ABB RobotStudio station: Station_[09.05.13]2.rsstn

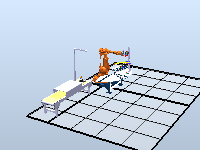
Station Station_[09.05.13] (saved by RobotStudio format 3)
Controller IRB2400_10kg_1.5m_3, task T_ROB1: task frame (RAPID world) sits at (0, 0, 226) mm in the station
Controller IRB2400_10kg_1.5m_3
  mechanical unit ROB_1: IRB2400_10_150__02, 6 joints, base frame (0, 0, -10) mm
Layout (positions relative to the parent item):
  - IRB2400_10_150__02 [mechanism, from Robots\IRB2400_10_150__02.rslib] at (0, 0, 216) mm; joint values [0, 0, 0, 0, 0, 0] (rad or m)
  - Table3_2 [part]
  - SC_RightDispenser [smart component] at (848.89, 660.39, 707) mm, rotated rx 0 ry 0 rz -142.5 deg
      signals: DI diNewPin, DO doPinInPosition2, DO doPinInPosition1
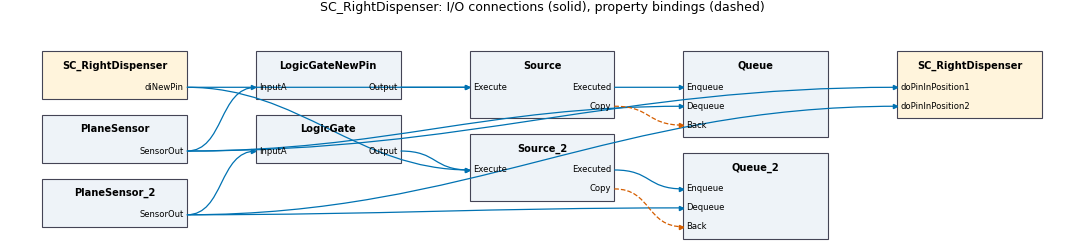
      connections:
        SC_RightDispenser.diNewPin -> Source.Execute
        Source.Executed -> Queue.Enqueue
        PlaneSensor.SensorOut -> Queue.Dequeue
        PlaneSensor.SensorOut -> SC_RightDispenser.doPinInPosition1
        PlaneSensor.SensorOut -> LogicGateNewPin.InputA
        LogicGateNewPin.Output -> Source.Execute
        SC_RightDispenser.diNewPin -> Source_2.Execute
        Source_2.Executed -> Queue_2.Enqueue
        PlaneSensor_2.SensorOut -> Queue_2.Dequeue
        PlaneSensor_2.SensorOut -> SC_RightDispenser.doPinInPosition2
        PlaneSensor_2.SensorOut -> LogicGate.InputA
        LogicGate.Output -> Source_2.Execute
        Source.Copy => Queue.Back
        Source_2.Copy => Queue_2.Back
    - Dispenser [part]
    - Source [smart component]
        properties: Source=Pin; Copy=Pin_291; Parent=(none); Position=[-0.078 0.0985 0.189]; Orientation=[0 0 0]; Transient=false
        signals: DI Execute, DO Executed
    - Queue [smart component]
        properties: Back=Pin_291; Front=(none); Queue={410cd2da-901c-4602-b1b9-b274db1111d8};{51c41708-d6a1-4a4a-81b2-86109b64f340};{5f0a7e8e-897b-4f59-8c9f-8c525d5b29a4};{57ea5d73-423b-4f0f-a570-9931c59fdda0};{5ccf77fa-e120-45a3-9187-0274426f82fc};{74150822-190d-40d8-916f-0fd6875921bc};{baa7ba2a-e563-400f-ae00-338ac9d6b310};{166c1fa7-f084-4893-8c68-a7378bc4935a};{0c8467ce-4cb3-4075-8f36-e6447ecc44ba};{a4931bd6-61c0-4022-957d-34420e4f6ad0};{b2f85a70-4d19-413a-b019-3afa180c1445};{512256d1-278f-462d-98f1-9ffcbd4d9afc};{849db594-4dfe-4c58-a8bd-451d21853566};{c968444c-bd1a-4f2f-bbaa-bfd3e7f50be5};{53c4b951-dfc2-4c08-b51d-efe4876241dc};{64f07cc2-7ba3-4255-a888-147bdde81c96};{5e5e12c0-75f5-4fd7-8049-5710cdd06950};{7bc2919c-0f2a-489c-9e4c-df3bff6561ed};{5aa4b278-0833-4ca9-af8d-253aa8523874};{1baac950-fc54-4ea7-852c-7f888843f6f9};{b4b16473-bd2b-40f5-a110-90fbcba822d9};{d003a69b-5307-4c56-b226-d498155ba824};{d659394f-77c7-41ee-9797-cd61472f6401};{a8294731-aa9f-4324-81a7-55ebbef1ff1c};{1eff712e-2c63-4fa8-99b0-fad1482486d3};{b15f9735-19cd-4f7a-8d4f-e540a16427f5};{02485707-3f80-4cc3-94a6-af0fe382acfb};{ec0e8ce0-b480-4ff5-b740-0a7d244ffb35};{21e78636-7eb3-4061-8dde-926c3e464303};{0772fef3-b80e-464b-9cad-322a585d167a};{d8ed8ead-e522-4938-9c7c-7997e1d5aae1};{4dfefca0-2913-4484-9455-684dfc1cbf5a};{f8c8569f-a97f-4f57-84f0-3da59c0f2755};{9fd95979-e5cf-4fa7-b177-2c560699c82c};{84f56170-3294-4345-a728-b2bfe69be833};{b3710d51-6f0f-48ac-9b0f-811ac7c7d083};{c8300349-23e3-4531-beb4-4210900096fb}; NumberOfObjects=0
        signals: DI Enqueue, DI Dequeue, DI Clear, DI Delete, DI DeleteAll
    - LinearMover [smart component]
        properties: Object=Queue; Direction=[0 0 -0.07]; Speed=0.05; Reference=Global; ReferenceObject=(none)
        signals: DI Execute
    - PlaneSensor [smart component]
        properties: Origin=[-0.0530000000000006 0.1235 0.1195]; Axis1=[-0.03 0 0]; Axis2=[0 -0.04 0]; SensedPart=Pin_291
        signals: DI Active, DO SensorOut
      - _sensorPart_ [part]
    - Pin [part] at (-78, 98.5, 189) mm
    - LogicGateNewPin [smart component]
        properties: Operator=NOT; Delay=0
        signals: DI InputA, DI InputB, DO Output
    - Source_2 [smart component]
        properties: Source=Pin_2; Copy=Pin_2_290; Parent=(none); Position=[-0.078 -0.0985 0.198]; Orientation=[0 0 0]; Transient=false
        signals: DI Execute, DO Executed
    - Queue_2 [smart component]
        properties: Back=Pin_2_290; Front=(none); Queue={9b8a8857-6c8e-4b14-9da2-826ab751c38e};{88bba264-885b-495e-9113-affa9235d31d};{50c1a2e4-cd05-4fea-a5f8-244e054fca82};{1c26a820-5f81-4fc8-b661-270a696b215b};{079caa1e-4b65-4731-ac2d-b38991013e84};{04249497-c8e4-4d2b-8d23-0d0c3b1232f2};{9b46111e-8043-4ec7-820f-f6b1f3216e0a};{190405bf-72c0-4a75-968d-0e05791ba659};{cdaa2867-23d2-4f9c-8306-ddafce1e9ac9};{a0d1b5cc-bcdc-4e7d-b91f-09bc5bc174e5};{802900b3-44c0-4e10-9d61-adfd75a0d86d};{e1828195-6a4a-4e48-b78f-f1287aff9cdc};{27d5d252-1980-452a-aff5-49173c411714};{b44ede4c-8dd3-43ce-8da4-3f1fb091dc7f};{168b000f-829e-439e-a2b5-5bc5735400ce};{aacdfd62-2178-4132-b345-2cd6db76197d};{33bd895a-7dcf-445c-8a77-0a7b01e583dc};{c1a42cbc-38c3-48e5-a615-b149ac9d8780};{fcea76f5-b349-47ef-a520-1d1e9307533b};{d936eec8-07d3-4a18-b33b-be549f4009da};{161ff837-8ce6-447d-8217-59dc5e5add53}; NumberOfObjects=0
        signals: DI Enqueue, DI Dequeue, DI Clear, DI Delete, DI DeleteAll
    - LinearMover_2 [smart component]
        properties: Object=Queue_2; Direction=[0 0 -0.07]; Speed=0.05; Reference=Global; ReferenceObject=(none)
        signals: DI Execute
    - PlaneSensor_2 [smart component]
        properties: Origin=[-0.053 -0.1235 0.1195]; Axis1=[-0.03 0 0]; Axis2=[0 0.04 0]; SensedPart=Pin_2_290
        signals: DI Active, DO SensorOut
      - _sensorPart_ [part]
    - LogicGate [smart component]
        properties: Operator=NOT; Delay=0
        signals: DI InputA, DI InputB, DO Output
    - Pin_2 [part] at (-78, -98.5, 189) mm
    - Pin_2_290 [part] at (-78, -98.5, 118.8) mm
    - Pin_291 [part] at (-78, 98.5, 119.4) mm
  - SC_Conveyor[190413] [smart component] at (45.5, -3634, 0) mm
      signals: DI diPalletOut, DI diPalletIn, DO doPalletAtEnd, DO doPalletAtStart, DO diPalletMovingOut, DO doPalletMovingIn, DI diConDir, DI diConRun
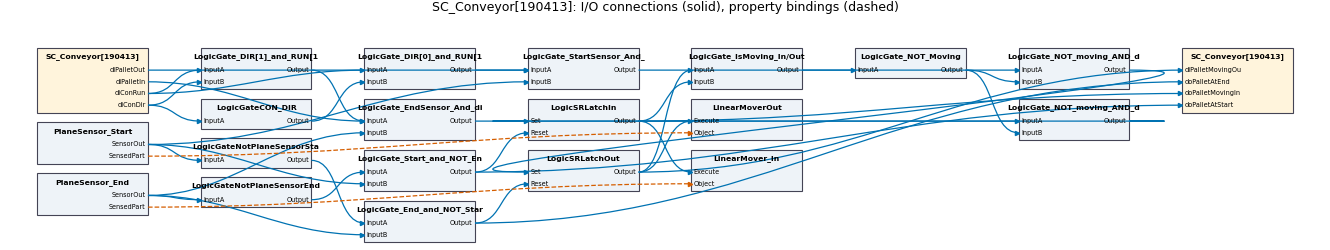
      connections:
        SC_Conveyor[190413].diPalletOut -> LogicGate_StartSensor_And_diOUT.InputA
        PlaneSensor_Start.SensorOut -> LogicGate_StartSensor_And_diOUT.InputB
        PlaneSensor_Start.SensorOut -> LogicGateNotPlaneSensorStart.InputA
        LogicGate_StartSensor_And_diOUT.Output -> LogicGate_NOT_moving_AND_diOUT.InputA
        LogicGate_NOT_Moving.Output -> LogicGate_NOT_moving_AND_diOUT.InputB
        LogicGate_NOT_moving_AND_diOUT.Output -> LogicSRLatchOut.Set
        LogicSRLatchOut.Output -> LinearMoverOut.Execute
        LogicSRLatchOut.Output -> SC_Conveyor[190413].diPalletMovingOut
        LogicGateNotPlaneSensorStart.Output -> LogicGate_End_and_NOT_Start.InputA
        PlaneSensor_End.SensorOut -> LogicGate_End_and_NOT_Start.InputB
        LogicGate_End_and_NOT_Start.Output -> LogicSRLatchOut.Reset
        LogicGate_End_and_NOT_Start.Output -> SC_Conveyor[190413].doPalletAtEnd
        SC_Conveyor[190413].diPalletIn -> LogicGate_EndSensor_And_diIN.InputA
        PlaneSensor_End.SensorOut -> LogicGate_EndSensor_And_diIN.InputB
        PlaneSensor_End.SensorOut -> LogicGateNotPlaneSensorEnd.InputA
        LogicGate_EndSensor_And_diIN.Output -> LogicGate_NOT_moving_AND_diIN.InputA
        LogicGate_NOT_Moving.Output -> LogicGate_NOT_moving_AND_diIN.InputB
        LogicGate_NOT_moving_AND_diIN.Output -> LogicSRLatchIn.Set
        LogicSRLatchIn.Output -> LinearMover_In.Execute
        LogicSRLatchIn.Output -> SC_Conveyor[190413].doPalletMovingIn
        LogicGateNotPlaneSensorEnd.Output -> LogicGate_Start_and_NOT_End.InputA
        PlaneSensor_Start.SensorOut -> LogicGate_Start_and_NOT_End.InputB
        LogicGate_Start_and_NOT_End.Output -> LogicSRLatchIn.Reset
        LogicGate_Start_and_NOT_End.Output -> SC_Conveyor[190413].doPalletAtStart
        LogicSRLatchOut.Output -> LogicGate_IsMoving_In/Out.InputA
        LogicSRLatchIn.Output -> LogicGate_IsMoving_In/Out.InputB
        LogicGate_IsMoving_In/Out.Output -> LogicGate_NOT_Moving.InputA
        SC_Conveyor[190413].diConRun -> LogicGate_DIR[0]_and_RUN[1].InputA
        SC_Conveyor[190413].diConDir -> LogicGateCON_DIR.InputA
        LogicGateCON_DIR.Output -> LogicGate_DIR[0]_and_RUN[1].InputB
        LogicGate_DIR[0]_and_RUN[1].Output -> LogicGate_StartSensor_And_diOUT.InputA
        SC_Conveyor[190413].diConRun -> LogicGate_DIR[1]_and_RUN[1].InputA
        SC_Conveyor[190413].diConDir -> LogicGate_DIR[1]_and_RUN[1].InputB
        LogicGate_DIR[1]_and_RUN[1].Output -> LogicGate_EndSensor_And_diIN.InputA
        PlaneSensor_Start.SensedPart => LinearMoverOut.Object
        PlaneSensor_End.SensedPart => LinearMover_In.Object
    - Conveyor3 [part] at (0, 0, 606) mm
    - PlaneSensor_Start [smart component, from RobotStudio\SC_RightDispenser[080513].rslib]
        properties: Origin=[-0.05 0.4 0.62]; Axis1=[-0.5 0 0]; Axis2=[0 2.1 0]; SensedPart=Pallet
      - _sensorPart_ [part]
    - PlaneSensor_End [smart component, from RobotStudio\SC_RightDispenser[080513].rslib]
        properties: Origin=[-0.05 0 0.62]; Axis1=[-0.5 0 0]; Axis2=[0 2.2 0]; SensedPart=(none)
      - _sensorPart_ [part]
    - LinearMoverOut [smart component, from RobotStudio\SC_RightDispenser[080513].rslib]
        properties: Object=Pallet; Direction=[0 -1 0]; Speed=0.6; Reference=Global; ReferenceObject=(none)
    - LinearMover_In [smart component, from RobotStudio\SC_RightDispenser[080513].rslib]
        properties: Object=(none); Direction=[0 1 0]; Speed=0.6; Reference=Global; ReferenceObject=(none)
    - LogicGateNotPlaneSensorStart [smart component]
        properties: Operator=NOT; Delay=0
        signals: DI InputA, DI InputB, DO Output
    - LogicGateNotPlaneSensorEnd [smart component]
        properties: Operator=NOT; Delay=0
        signals: DI InputA, DI InputB, DO Output
    - LogicSRLatchOut [smart component]
        signals: DI Set, DI Reset, DO Output, DO InvOutput
    - LogicSRLatchIn [smart component]
        signals: DI Set, DI Reset, DO Output, DO InvOutput
    - LogicGate_End_and_NOT_Start [smart component]
        properties: Operator=AND; Delay=0
        signals: DI InputA, DI InputB, DO Output
    - LogicGate_StartSensor_And_diOUT [smart component]
        properties: Operator=AND; Delay=0
        signals: DI InputA, DI InputB, DO Output
    - LogicGate_Start_and_NOT_End [smart component]
        properties: Operator=AND; Delay=0
        signals: DI InputA, DI InputB, DO Output
    - LogicGate_EndSensor_And_diIN [smart component]
        properties: Operator=AND; Delay=0
        signals: DI InputA, DI InputB, DO Output
    - LogicGate_IsMoving_In/Out [smart component]
        properties: Operator=OR; Delay=0
        signals: DI InputA, DI InputB, DO Output
    - LogicGate_NOT_Moving [smart component]
        properties: Operator=NOT; Delay=0
        signals: DI InputA, DI InputB, DO Output
    - LogicGate_NOT_moving_AND_diOUT [smart component]
        properties: Operator=AND; Delay=0
        signals: DI InputA, DI InputB, DO Output
    - LogicGate_NOT_moving_AND_diIN [smart component]
        properties: Operator=AND; Delay=0
        signals: DI InputA, DI InputB, DO Output
    - LogicGateCON_DIR [smart component]
        properties: Operator=NOT; Delay=0
        signals: DI InputA, DI InputB, DO Output
    - LogicGate_DIR[0]_and_RUN[1] [smart component]
        properties: Operator=AND; Delay=0
        signals: DI InputA, DI InputB, DO Output
    - LogicGate_DIR[1]_and_RUN[1] [smart component]
        properties: Operator=AND; Delay=0
        signals: DI InputA, DI InputB, DO Output
  - LogicGate [smart component]
      properties: Operator=NOT; Delay=0
      signals: DI InputA, DI InputB, DO Output
  - NewSmartGripper[040513] [smart component, from RobotStudio\NewSmartGripper[040513].rslib] at (940, 0, 1671) mm, rotated rx 0 ry 90 rz 0 deg
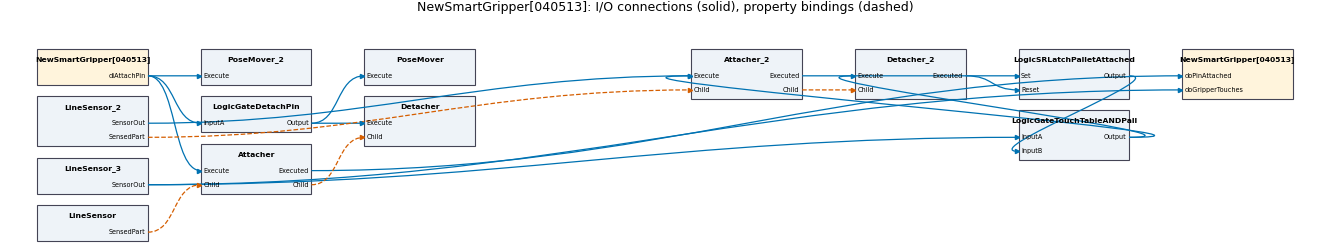
      connections:
        NewSmartGripper[040513].diAttachPin -> PoseMover_2.Execute
        NewSmartGripper[040513].diAttachPin -> Attacher.Execute
        NewSmartGripper[040513].diAttachPin -> LogicGateDetachPin.InputA
        LogicGateDetachPin.Output -> Detacher.Execute
        LogicGateDetachPin.Output -> PoseMover.Execute
        Attacher.Executed -> NewSmartGripper[040513].doPinAttached
        LineSensor_2.SensorOut -> Attacher_2.Execute
        Attacher_2.Executed -> LogicSRLatchPalletAttached.Set
        LineSensor_3.SensorOut -> NewSmartGripper[040513].doGripperTouchesTable
        LogicGateTouchTableANDPallet.Output -> Attacher_2.Execute
        LineSensor_3.SensorOut -> LogicGateTouchTableANDPallet.InputA
        LogicSRLatchPalletAttached.Output -> LogicGateTouchTableANDPallet.InputB
        LogicGateTouchTableANDPallet.Output -> Detacher_2.Execute
        Detacher_2.Executed -> LogicSRLatchPalletAttached.Reset
        LineSensor.SensedPart => Attacher.Child
        Attacher.Child => Detacher.Child
        LineSensor_2.SensedPart => Attacher_2.Child
        Attacher_2.Child => Detacher_2.Child
    - Attacher [smart component]
        properties: Parent=Attacher_2; Flange=1; Child=(none); Mount=false; Offset=[0 0 0]; Orientation=[0 0 0]
        signals: DI Execute, DO Executed
    - Attacher_2 [smart component]
        properties: Parent=Detacher; Flange=0; Child=(none); Mount=false; Offset=[0 0 0]; Orientation=[0 0 0]
        signals: DI Execute, DO Executed
    - Detacher [smart component]
        properties: Child=(none); KeepPosition=true
        signals: DI Execute, DO Executed
    - Detacher_2 [smart component]
        properties: Child=(none); KeepPosition=true
        signals: DI Execute, DO Executed
    - LineSensor [smart component]
        properties: Start=[0.03 0 0.1702]; End=[0.03 0 0.16]; Radius=0.002; SensedPart=(none); SensedPoint=[0 0 0]
        signals: DI Active, DO SensorOut
      - _sensorPart_ [part, from RobotStudio\NewSmartGripper[040513].rslib]
    - LineSensor_2 [smart component]
        properties: Start=[-0.109 0.07175 0.18]; End=[-0.109 0.07175 0.1]; Radius=0.0012; SensedPart=(none); SensedPoint=[0 0 0]
        signals: DI Active, DO SensorOut
      - _sensorPart_ [part, from RobotStudio\NewSmartGripper[040513].rslib]
    - LineSensor_3 [smart component]
        properties: Start=[-0.142 0 0.04]; End=[-0.12 0 0.04]; Radius=0.004; SensedPart=(none); SensedPoint=[0 0 0]
        signals: DI Active, DO SensorOut
      - _sensorPart_ [part, from RobotStudio\NewSmartGripper[040513].rslib]
    - PoseMover [smart component]
        properties: Mechanism=NewGripperMech; Pose=3; Duration=0.2
        signals: DI Execute, DI Pause, DI Cancel, DO Executed, DO Executing, DO Paused
    - PoseMover_2 [smart component]
        properties: Mechanism=NewGripperMech; Pose=2; Duration=0.2
        signals: DI Execute, DI Pause, DI Cancel, DO Executed, DO Executing, DO Paused
    - NewGripperMech [mechanism, from RobotStudio\NewSmartGripper[040513].rslib] at (0, 0, 0) mm; joint values [0, 0] (rad or m)
    - LogicGateDetachPin [smart component]
        properties: Operator=NOT; Delay=0
        signals: DI InputA, DI InputB, DO Output
    - LogicSRLatchPalletAttached [smart component, from Components\LogicSRLatch.rslib]
    - LogicGateTouchTableANDPallet [smart component]
        properties: Operator=AND; Delay=0
        signals: DI InputA, DI InputB, DO Output
  - Pallet [part] at (-346.06, -1163.98, 605.84) mm, rotated rx 0 ry -0.05 rz -90.02 deg
  - Frame_1 [frame] at (710.04, 677.11, 1017.54) mm, rotated rx -135.34 ry 89.95 rz -97.28 deg
Attachment: NewSmartGripper[040513] is attached to IRB2400_10_150__02 / Link6
EventTableEntry 5: Group=, Trigger=Grip 6, Actions=[diGRIP 7], Comment=, ActivationMode=2, Cyclic=false
EventTableTriggerIO 6: IOValue=[1], IRC5Controller=? -1, Operator=0, SignalSource=IRB2400_10kg_1.5m_3 486
EventTableActionIO 7: IOValue=[0], IRC5Controller=? -1, SignalTarget=Station_[09.05.13] 1
EventTableEntry 8: Group=, Trigger=Grip 9, Actions=[diGRIP 10], Comment=, ActivationMode=2, Cyclic=false
EventTableTriggerIO 9: IOValue=[0], IRC5Controller=? -1, Operator=0, SignalSource=IRB2400_10kg_1.5m_3 486
EventTableActionIO 10: IOValue=[1], IRC5Controller=? -1, SignalTarget=Station_[09.05.13] 1
EventTableTriggerIO 1726: IOValue=[1], IRC5Controller=? -1, Operator=0, SignalSource=IRB2400_10kg_1.5m_3 486
EventTableTriggerIO 1727: IOValue=[0], IRC5Controller=? -1, Operator=0, SignalSource=IRB2400_10kg_1.5m_3 486
EventTableEntry 1775: Group=, Trigger=ConRun 1776, Actions=[diStationConRun 1777], Comment=, ActivationMode=2, Cyclic=false
EventTableTriggerIO 1776: IOValue=[1], IRC5Controller=? -1, Operator=0, SignalSource=IRB2400_10kg_1.5m_3 486
EventTableActionIO 1777: IOValue=[1], IRC5Controller=? -1, SignalTarget=Station_[09.05.13] 1
EventTableEntry 1778: Group=, Trigger=ConDir 1779, Actions=[diStationConDir 1780], Comment=, ActivationMode=2, Cyclic=false
EventTableTriggerIO 1779: IOValue=[1], IRC5Controller=? -1, Operator=0, SignalSource=IRB2400_10kg_1.5m_3 486
EventTableActionIO 1780: IOValue=[1], IRC5Controller=? -1, SignalTarget=Station_[09.05.13] 1
EventTableEntry 1781: Group=, Trigger=ConRun 1782, Actions=[diStationConRun 1783], Comment=, ActivationMode=2, Cyclic=false
EventTableTriggerIO 1782: IOValue=[0], IRC5Controller=? -1, Operator=0, SignalSource=IRB2400_10kg_1.5m_3 486
EventTableActionIO 1783: IOValue=[0], IRC5Controller=? -1, SignalTarget=Station_[09.05.13] 1
EventTableEntry 1784: Group=, Trigger=ConDir 1785, Actions=[diStationConDir 1786], Comment=, ActivationMode=2, Cyclic=false
EventTableTriggerIO 1785: IOValue=[0], IRC5Controller=? -1, Operator=0, SignalSource=IRB2400_10kg_1.5m_3 486
EventTableActionIO 1786: IOValue=[0], IRC5Controller=? -1, SignalTarget=Station_[09.05.13] 1
Station signals: DI diRunConOUT, DI diRunConIN, DI diGRIP, DI diNewPinINDISP, DI diStationConRun, DI diStationConDir
Station logic (signal -> signal, property => property):
  Station_[09.05.13].diGRIP -> NewSmartGripper[040513].diAttachPin
  Station_[09.05.13].diNewPinINDISP -> SC_RightDispenser.diNewPin
  Station_[09.05.13].diStationConRun -> SC_Conveyor[190413].diConRun
  Station_[09.05.13].diStationConDir -> SC_Conveyor[190413].diConDir
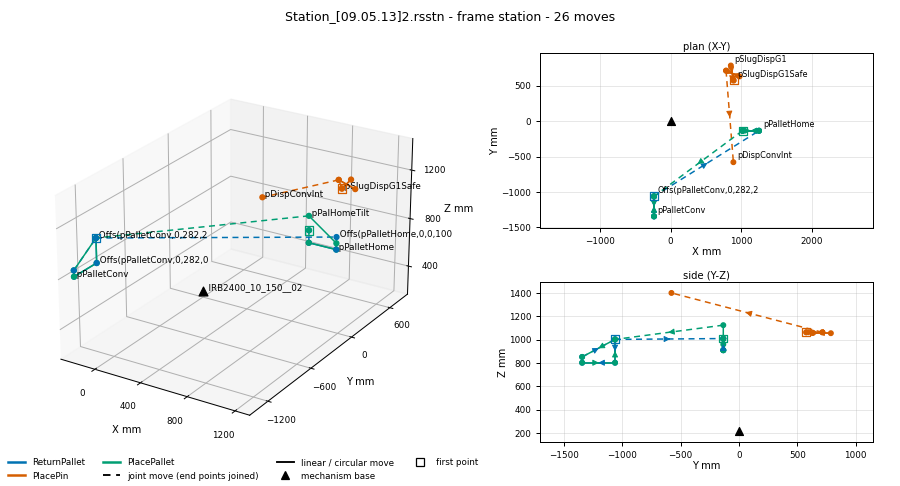
[picture p0: tool path of Station_[09.05.13]2.rsstn in frame station, 26 of 38 moves have a stored position in this frame; points joined in program order, loops and branches not executed]
Targets, tools, work objects and paths stored in the station, written as RAPID:
! task T_ROB1
MODULE MW
  PERS tooldata tGrip:=[TRUE,[[30,0,180],[1,0,0,0]],[1.5,[0,0,80],[1,0,0,0],0,0,0]];
  PERS tooldata tTine:=[TRUE,[[-114.5,0,234.15],[1,0,0,0]],[1.5,[0,0,80],[1,0,0,0],0.04,0.04,0.04]];
  CONST robtarget pPalletConv:=[[-234.56,-1344.02,576.85],[0.500039998,0.499942998,-0.500039998,0.499976998],[-2,-1,-2,0],[9E9,9E9,9E9,9E9,9E9,9E9]];
  CONST robtarget pPalletHome:=[[1250.04,-133.95,684.28],[0.000048,-0.707407715,-0.000048,-0.706805716],[-1,-1,-2,0],[9E9,9E9,9E9,9E9,9E9,9E9]];
  CONST jointtarget jtCalibPos:=[[0,0,0,0,0,0],[9E9,9E9,9E9,9E9,9E9,9E9]];
  CONST robtarget pSlugDispG1Safe:=[[890.6,577.3,837.9],[0.678140503,-0.200710149,0.678000503,0.200390149],[0,0,-1,0],[9E9,9E9,9E9,9E9,9E9,9E9]];
  CONST robtarget pSlugDispG1:=[[851.75,788.07,830.08],[0.668320736,-0.230855909,0.668581736,0.230328909],[0,0,-1,0],[9E9,9E9,9E9,9E9,9E9,9E9]];
  CONST robtarget pSlugDispG2Safe:=[[784.1,715.6,837.7],[0.658308518,-0.269043481,0.654098463,0.257683334],[0,-1,0,0],[9E9,9E9,9E9,9E9,9E9,9E9]];
  CONST robtarget pSlugDispG2:=[[974.96,633.73,831.83],[0.668405716,-0.230831902,0.668514716,0.230300902],[0,-1,0,0],[9E9,9E9,9E9,9E9,9E9,9E9]];
  CONST robtarget pDispConvInt:=[[887.7,-578.4,1175.2],[0.654679605,0.26514984,0.656439604,-0.26490984],[-1,-1,0,0],[9E9,9E9,9E9,9E9,9E9,9E9]];
  CONST robtarget pPalHomeTilt:=[[1015.987042359,-133.981901811,898.978895592],[0.000045049,-0.665857682,-0.00005045,-0.746078778],[-1,-1,-2,0],[9E9,9E9,9E9,9E9,9E9,9E9]];
  PROC main()
  ENDPROC
  PROC ReturnPallet()
    MoveJ Offs(pPalletConv,0,282,200),v1000,fine,tTine;
    MoveL Offs(pPalletConv,0,282,0),v200,fine,tTine;
    MoveL pPalletConv,v200,fine,tTine;
    MoveL Offs(pPalletConv, 0,0,50),v200,fine,tTine;
    MoveJ Offs(pPalletConv,0,282,200),v1000,fine,tTine;
    MoveJ Offs(pPalletHome,0,0,100),v1000,fine,tTine;
    MoveL pPalletHome,v200,fine,tTine;
    MoveL Offs(pPalletHome,-232,0,0),v500,fine,tTine;
    MoveJ Offs(pPalletHome,-232,0,100),v1000,fine,tTine;
    MoveAbsJ jtCalibPos,v1000,fine,tTine;
  ENDPROC
  PROC RemovePin()
    MoveJ Offs(pSlugPallConvCD,0,0,100),v1000,fine,tGrip;
    Set Grip;
    MoveL Offs(pSlugPallH1G, xoffset, yoffset, 50),v200,fine,tGrip;
    MoveL Offs(pSlugPallH1G, xoffset, yoffset, 0),v200,fine,tGrip;
    Reset Grip;
    WaitTime 1;
    MoveL Offs(pSlugPallH1G, xoffset, yoffset, 200),v200,fine,tGrip;
    MoveAbsJ jtCalibPos,v1000,fine,tTine;
    Reset Grip;
  ENDPROC
  PROC PlacePin()
    MoveJ pSlugDispG1Safe,v500,fine,tGrip;
    MoveL pSlugDispG1,v200,fine,tGrip;
    Set Grip;
    WaitTime 1;
    MoveL pSlugDispG1Safe,v200,fine,tGrip;
    MoveJ pSlugDispG2Safe,v1000,fine,tGrip;
    MoveL pSlugDispG2,v200,fine,tGrip;
    Set Grip;
    WaitTime 1;
    MoveL pSlugDispG2Safe,v200,fine,tGrip;
    MoveJ pDispConvInt,v1000,fine,tGrip;
    MoveJ Offs(pSlugPallConvCD,0,0,200),v1000,fine,tGrip;
    MoveL Offs(pSlugPallH1D, xoffset, yoffset, 50),v200,fine,tGrip;
    MoveL Offs(pSlugPallH1D, xoffset, yoffset, 0),v200,fine,tGrip;
    Reset Grip;
    WaitTime 1;
    MoveL Offs(pSlugPallH1D, xoffset, yoffset, 100),v200,fine,tGrip;
    MoveAbsJ jtCalibPos,v1000,fine,tTine;
  ENDPROC
  PROC PlacePallet()
    MoveJ Offs(pPalletHome,-232,0,100),v1000,fine,tTine;
    MoveJ Offs(pPalletHome,-232,0,0),v500,fine,tTine;
    MoveL pPalletHome,v200,fine,tTine;
    MoveL Offs(pPalletHome,0,0,50),v200,fine,tTine;
    MoveL pPalHomeTilt,v200,fine,tTine;
    MoveJ Offs(pPalletConv,0,282,200),v1000,fine,tTine;
    MoveL Offs(pPalletConv,0,0,50),v500,fine,tTine;
    MoveL pPalletConv,v200,fine,tTine;
    MoveL Offs(pPalletConv,0,282,0),v200,fine,tTine;
    MoveL Offs(pPalletConv,0,282,200),v500,fine,tTine;
    MoveAbsJ jtCalibPos,v1000,fine,tTine;
  ENDPROC
ENDMODULE

! task T_ROB1
MODULE CalibData
  PERS tooldata Tooldata_1:=[TRUE,[[20,0,175.76],[0.707106781,0,-0.707106781,0]],[1,[0,0,1],[1,0,0,0],0,0,0]];
  PERS tooldata Tooldata_2:=[TRUE,[[-83.5,0,233],[0,0.707106781,0,0.707106781]],[1,[0,0,1],[1,0,0,0],0,0,0]];
  PERS tooldata My_Mechanism_1:=[TRUE,[[20,0,175.76],[0.707106781,0,-0.707106781,0]],[1,[0,0,1],[1,0,0,0],0,0,0]];
  PERS tooldata My_Mechanism_2:=[TRUE,[[-83.5,0,233],[0,0.707106781,0,0.707106781]],[1,[0,0,1],[1,0,0,0],0,0,0]];
ENDMODULE

